# EPICS alarm handler configuration: apps/alh/HPS.alhConfig
#===============================================================================
# HPS Top-level Alarm Config
#===============================================================================

GROUP    NULL                         HPS

$GUIDANCE
    For info on target-related items, please contact HPS Experts
$END

#=======================================
# Subsystems
#=======================================

INCLUDE HPS /usr/clas12/hps/prod/apps/alh/beam.alhConfig
INCLUDE HPS /usr/clas12/hps/prod/apps/alh/ecal.alhConfig
INCLUDE HPS /usr/clas12/hps/prod/apps/alh/fcup.alhConfig
